// TIA Portal project "PRT" (V13)

(* hardware
DEVICE "S7300/ET200M-Station_1"  S7-300 station
   slot 0: "Profilschiene_0"  Rail  6ES7 390-1***0-0AA0
   slot 1: "PS 307 5A_1"  PS 307 5A  6ES7 307-1EA00-0AA0
   slot 2: "SIMATIC S7-300"  CPU 314C-2 PN/DP  6ES7 314-6EH04-0AB0  V3.3
      slot 2: "PROFINET-Schnittstelle_1"  PN-IO
         slot 1: "Port_1"  Port
         slot 2: "Port_2"  Port
      slot 5: "DI 24/DO 16_1"  DI24/DO16
      slot 6: "AI 5/AO 2_1"  AI5/AO2
      slot 7: "Zählen_1"  Counter
      slot 8: "Positionieren_1"  Positioning
   slot 4: "CP 343-2_1"  CP 343-2  6GK7 343-2AH01-0XA0  V3.1
*)

// ===== PLC "SIMATIC S7-300"  CPU 314C-2 PN/DP =====

VAR_GLOBAL   // PLC tag table "Standard-Variablentabelle"
   "Ix_S1_Start" AT %I124.0 : Bool;   // Start pushbutton
   "Ix_1B2_CylA1Ext" AT %I124.1 : Bool;   // Cylinder 1A1 extended
   "Ix_2B2_CylA2Ext" AT %I124.2 : Bool;   // Cylinder 2A1 extended
   "Mx_Step0" AT %M10.0 : Bool;   // Grafcet, step-flag 0
   "Mx_Step1" AT %M10.1 : Bool;   // Grafcet, step-flag 1
   "Mx_Step2" AT %M10.2 : Bool;   // Grafcet, step-flag 2
   "Mx_Step3" AT %M10.3 : Bool;   // Grafcet, step-flag 3
   "Mx_Step4" AT %M10.4 : Bool;   // Grafcet, step-flag4
   "Mx_StartingFlag" AT %M20.0 : Bool;   // Starting flag to activate the sequence ( Step 0)
   "Qx_1M1_MoveCyl1A1Out" AT %Q124.0 : Bool;   // Move cylinder 1A1 out
   "Qx_1M1_MoveCyl1A1In" AT %Q124.1 : Bool;   // Move cylinder 1A1 in
   "Qx_1M1_MoveCyl2A1Out" AT %Q124.2 : Bool;   // Move cylinder 2A1
   "Mb_FlagByte10" AT %MB10 : Byte;   // Flag byte 10
   "Mb_FlagByte20" AT %MB20 : Byte;   // Flag byte 20
END_VAR

FUNCTION "Grafcet" : Void   // FC1, FBD
{ S7_Optimized_Access := 'FALSE' }
VERSION : 0.1
BEGIN

REGION Network 1: Step 0
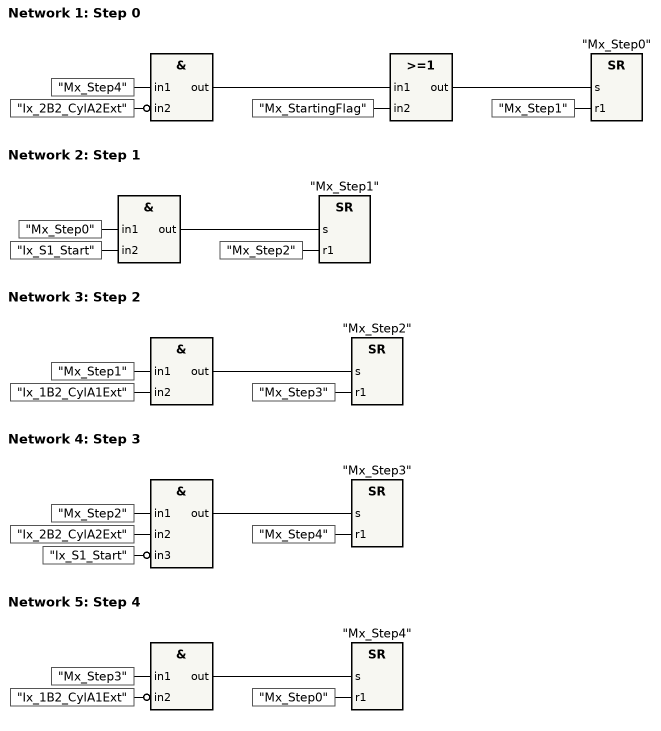
   IF ("Mx_Step4" AND NOT "Ix_2B2_CylA2Ext") OR "Mx_StartingFlag" THEN
       "Mx_Step0" := TRUE;   // SR flip-flop
   END_IF;
   IF "Mx_Step1" THEN "Mx_Step0" := FALSE; END_IF;
END_REGION

REGION Network 2: Step 1
   IF "Mx_Step0" AND "Ix_S1_Start" THEN
       "Mx_Step1" := TRUE;   // SR flip-flop
   END_IF;
   IF "Mx_Step2" THEN "Mx_Step1" := FALSE; END_IF;
END_REGION

REGION Network 3: Step 2
   IF "Mx_Step1" AND "Ix_1B2_CylA1Ext" THEN
       "Mx_Step2" := TRUE;   // SR flip-flop
   END_IF;
   IF "Mx_Step3" THEN "Mx_Step2" := FALSE; END_IF;
END_REGION

REGION Network 4: Step 3
   IF "Mx_Step2" AND "Ix_2B2_CylA2Ext" AND NOT "Ix_S1_Start" THEN
       "Mx_Step3" := TRUE;   // SR flip-flop
   END_IF;
   IF "Mx_Step4" THEN "Mx_Step3" := FALSE; END_IF;
END_REGION

REGION Network 5: Step 4
   IF "Mx_Step3" AND NOT "Ix_1B2_CylA1Ext" THEN
       "Mx_Step4" := TRUE;   // SR flip-flop
   END_IF;
   IF "Mx_Step0" THEN "Mx_Step4" := FALSE; END_IF;
END_REGION
END_FUNCTION

FUNCTION "Actions" : Void   // FC2, FBD
{ S7_Optimized_Access := 'FALSE' }
VERSION : 0.1
BEGIN

REGION Network 1: Move cylinder 1A1 out
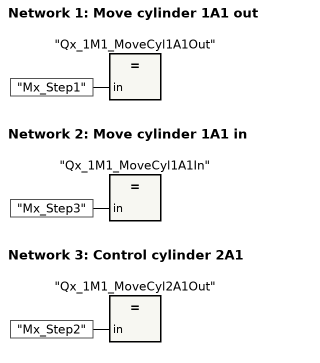
   "Qx_1M1_MoveCyl1A1Out" := "Mx_Step1";
END_REGION

REGION Network 2: Move cylinder 1A1 in
   "Qx_1M1_MoveCyl1A1In" := "Mx_Step3";
END_REGION

REGION Network 3: Control cylinder 2A1
   "Qx_1M1_MoveCyl2A1Out" := "Mx_Step2";
END_REGION
END_FUNCTION

ORGANIZATION_BLOCK "Main"   // OB1, FBD
TITLE = "Main Program Sweep (Cycle)"
{ S7_Optimized_Access := 'FALSE' }
VERSION : 0.1
BEGIN

REGION Network 1: Call the funciton diagram block
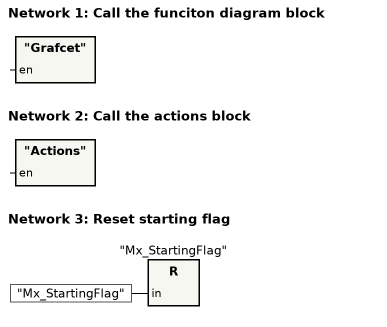
   "Grafcet"();
END_REGION

REGION Network 2: Call the actions block
   "Actions"();
END_REGION

REGION Network 3: Reset starting flag
   IF "Mx_StartingFlag" THEN "Mx_StartingFlag" := FALSE; END_IF;
END_REGION
END_ORGANIZATION_BLOCK

ORGANIZATION_BLOCK "COMPLETE RESTART"   // OB100, FBD
TITLE = "Complete Restart"
{ S7_Optimized_Access := 'FALSE' }
VERSION : 0.1
BEGIN

REGION Network 1: Reset flag byte number 10
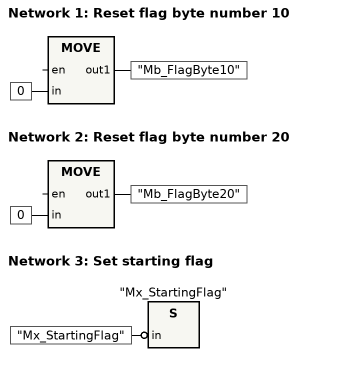
   "Mb_FlagByte10" := 0;
END_REGION

REGION Network 2: Reset flag byte number 20
   "Mb_FlagByte20" := 0;
END_REGION

REGION Network 3: Set starting flag
   IF NOT "Mx_StartingFlag" THEN "Mx_StartingFlag" := TRUE; END_IF;
END_REGION
END_ORGANIZATION_BLOCK